// TIA Portal V20 export
FUNCTION_BLOCK "LER_EQP_Interface"   // FB170, LAD
// stored: Access Published, MemoryReserve 100, SetENOAutomatically false
   VAR_INPUT
      enable : Bool;
      heartBeat : Byte;
      unitStatus : "LAF_typeUnitStatus";
      unitAlarms : "LAF_typeAlarms";
      partData : "LER_typePartData";
   END_VAR
   VAR_IN_OUT
      StackCommunication : "LER_typeCommunication";
      configuration : "LER_typeCommunicationConfiguration";
      moduleInterface : "LER_typeCommunicationInterface";
      controlNode : "LER_typeCommunicationControlNode";
   END_VAR
   VAR
      instEQP_Interface_Communication { S7_SetPoint := 'True'} : "LER_EQP_Communication";
   END_VAR
BEGIN

REGION Network 1: EQP Interface Suspend Command
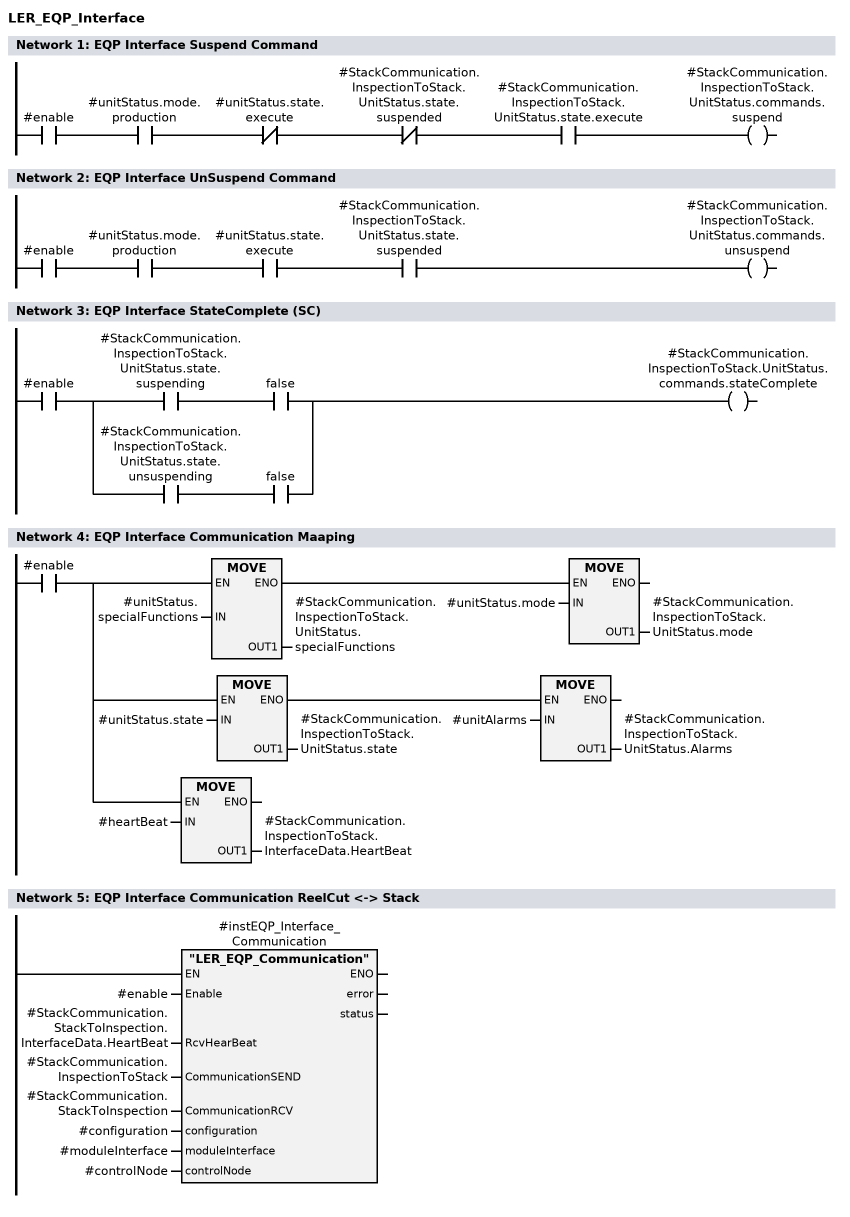
   RUNG wire#powerrail
      Contact( #enable )
      Contact( #unitStatus.mode.production )
      I_Contact( #unitStatus.state.execute )
      I_Contact( #StackCommunication.InspectionToStack.UnitStatus.state.suspended )
      Contact( #StackCommunication.InspectionToStack.UnitStatus.state.execute )
      Coil( #StackCommunication.InspectionToStack.UnitStatus.commands.suspend )
   END_RUNG
   // the same network as SCL:
   #StackCommunication.InspectionToStack.UnitStatus.commands.suspend := #enable AND #unitStatus.mode.production AND NOT #unitStatus.state.execute AND NOT #StackCommunication.InspectionToStack.UnitStatus.state.suspended AND #StackCommunication.InspectionToStack.UnitStatus.state.execute;
END_REGION

REGION Network 2: EQP Interface UnSuspend Command
   RUNG wire#powerrail
      Contact( #enable )
      Contact( #unitStatus.mode.production )
      Contact( #unitStatus.state.execute )
      Contact( #StackCommunication.InspectionToStack.UnitStatus.state.suspended )
      Coil( #StackCommunication.InspectionToStack.UnitStatus.commands.unsuspend )
   END_RUNG
   // the same network as SCL:
   #StackCommunication.InspectionToStack.UnitStatus.commands.unsuspend := #enable AND #unitStatus.mode.production AND #unitStatus.state.execute AND #StackCommunication.InspectionToStack.UnitStatus.state.suspended;
END_REGION

REGION Network 3: EQP Interface StateComplete (SC)
   RUNG wire#powerrail
      Contact( #enable )
      wire#w1
      Contact( #StackCommunication.InspectionToStack.UnitStatus.state.suspending )
      Contact( false )
      wire#w2
      Coil( #StackCommunication.InspectionToStack.UnitStatus.commands.stateComplete )
   END_RUNG
   RUNG wire#w1
      Contact( #StackCommunication.InspectionToStack.UnitStatus.state.unsuspending )
      Contact( false )
   END_RUNG wire#w2
   // the same network as SCL:
   #StackCommunication.InspectionToStack.UnitStatus.commands.stateComplete := #enable AND ((#StackCommunication.InspectionToStack.UnitStatus.state.suspending AND false) OR (#StackCommunication.InspectionToStack.UnitStatus.state.unsuspending AND false));
END_REGION

REGION Network 4: EQP Interface Communication Maaping
   RUNG wire#powerrail
      Contact( #enable )
      wire#w1
      Move(in := #unitStatus.specialFunctions, out1 => #StackCommunication.InspectionToStack.UnitStatus.specialFunctions)
      Move(in := #unitStatus.mode, out1 => #StackCommunication.InspectionToStack.UnitStatus.mode)
   END_RUNG
   RUNG wire#w1
      Move(in := #unitStatus.state, out1 => #StackCommunication.InspectionToStack.UnitStatus.state)
      Move(in := #unitAlarms, out1 => #StackCommunication.InspectionToStack.UnitStatus.Alarms)
   END_RUNG
   RUNG wire#w1
      Move(in := #heartBeat, out1 => #StackCommunication.InspectionToStack.InterfaceData.HeartBeat)
   END_RUNG
   // the same network as SCL:
   IF #enable THEN
       #StackCommunication.InspectionToStack.UnitStatus.specialFunctions := #unitStatus.specialFunctions;
       #StackCommunication.InspectionToStack.UnitStatus.mode := #unitStatus.mode;
       #StackCommunication.InspectionToStack.UnitStatus.state := #unitStatus.state;
       #StackCommunication.InspectionToStack.UnitStatus.Alarms := #unitAlarms;
       #StackCommunication.InspectionToStack.InterfaceData.HeartBeat := #heartBeat;
   END_IF;
END_REGION

REGION Network 5: EQP Interface Communication ReelCut <-> Stack
   RUNG wire#powerrail
      #instEQP_Interface_Communication(Enable := #enable, RcvHearBeat := #StackCommunication.StackToInspection.InterfaceData.HeartBeat, CommunicationSEND := #StackCommunication.InspectionToStack, CommunicationRCV := #StackCommunication.StackToInspection, configuration := #configuration, moduleInterface := #moduleInterface, controlNode := #controlNode, error =>, status =>)
   END_RUNG
   // the same network as SCL:
   #instEQP_Interface_Communication(Enable := #enable,   // "LER_EQP_Communication"
                           RcvHearBeat := #StackCommunication.StackToInspection.InterfaceData.HeartBeat,
                           CommunicationSEND := #StackCommunication.InspectionToStack,
                           CommunicationRCV := #StackCommunication.StackToInspection,
                           configuration := #configuration,
                           moduleInterface := #moduleInterface,
                           controlNode := #controlNode);
END_REGION
END_FUNCTION_BLOCK
